{attribute addProperty BoxType "KL9528"}
{attribute addProperty Id "OverloadAT %I*BOOL000UndervoltageAT %I*BOOL000ResetAT %Q*BOOL000"}
{attribute addProperty CRC "1406782961"}
{attribute addProperty SizeInBites "0"}
{attribute addProperty SizeInBytes "0"}
TYPE Channel_53D9CDF1 :
STRUCT
	{attribute addProperty Name "Overload"}
	Overload AT %I* : BOOL;
	{attribute addProperty Name "Undervoltage"}
	Undervoltage AT %I* : BOOL;
	{attribute addProperty Name "Reset"}
	Reset AT %Q* : BOOL;
END_STRUCT
END_TYPE

(* stored: Version 1.2.0.0, ProductVersion 3.1.4024.9
   DUT Channel_53D9CDF1: Id {8bb14078-ec05-4bc0-b384-1d06f6ceb962} *)
